PROGRAM MAIN
VAR
END_VAR

END_PROGRAM

(* stored: Version 1.1.0.1
   POU MAIN: Id {f7e68bb5-7ff0-472d-9b98-b668b5a71acd} *)
